{attribute 'GeneratedUsingTerminal: EL7041-0000-0016'}
{attribute addProperty BoxType "EL7041-0000-0016"}
{attribute addProperty Id "ENC_Status_compactAT %I*ENC_Status_compact_4D066E1A16STM_StatusAT %I*STM_Status_36ED096F11ENC_Control_compactAT %Q*ENC_Control_compact_21E2D14D6STM_ControlAT %Q*STM_Control_5A8B50163STM_VelocityAT %Q*STM_Velocity_A47A3F412WcStateAT %I*WcState_9091E0EB2InfoDataAT %I*InfoData_81897D033"}
{attribute addProperty CRC "886233229"}
{attribute addProperty Size "43"}
TYPE EL7041_34D2D88D EXTENDS EtcSlaveTerminalBase_947E5A46 :
STRUCT
	{attribute addProperty Name "ENC_Status_compact"}
	ENC_Status_compact : ENC_Status_compact_4D066E1A;
	{attribute addProperty Name "STM_Status"}
	STM_Status : STM_Status_36ED096F;
	{attribute addProperty Name "ENC_Control_compact"}
	ENC_Control_compact : ENC_Control_compact_21E2D14D;
	{attribute addProperty Name "STM_Control"}
	STM_Control : STM_Control_5A8B5016;
	{attribute addProperty Name "STM_Velocity"}
	STM_Velocity : STM_Velocity_A47A3F41;
	{attribute addProperty Name "WcState"}
	WcState : WcState_9091E0EB;
	{attribute addProperty Name "InfoData"}
	InfoData : InfoData_81897D03;
END_STRUCT
END_TYPE

(* stored: Version 1.2.0.0, ProductVersion 3.1.4024.9
   DUT EL7041_34D2D88D: Id {e53834be-ad3f-4f2e-b83f-a530d68a63a2} *)
